// TIA Portal V18 export
TYPE "PresserRecipe"
// stored: IsFailsafeCompliant false
   STRUCT
      PressCurveStartPosUL : Real;   // 压装开始位移上限值
      PressCurveStartPosLL : Real;   // 压装开始位移下限值
      PressCurveStartForceUL : Real;   // 压装开始压力上限值
      PressCurveStartForceLL : Real;   // 压装开始压力下限值
      PressCurveMiddlePosUL : Real;   // 压装过程位移上限值
      PressCurveMiddlePosLL : Real;   // 压装过程位移下限值
      PressCurveMiddleForceUL : Real;   // 压装过程压力上限值
      PressCurveMiddleForceLL : Real;   // 压装过程压力下限值
      PressCurveFinalPosUL : Real;   // 压装最终位移上限值
      PressCurveFinalPosLL : Real;   // 压装最终位移下限值
      PressCurveFinalForceUL : Real;   // 压装最终压力上限值
      PressCurveFinalForceLL : Real;   // 压装最终压力下限值
      PresserProgramNum : Int;   // 压机程序号
   END_STRUCT;
END_TYPE
